# B&R Automation Studio project stopGate_FuB
Automation Studio 4.9

## Logical view

Binary libraries used (declarations not repeated): operator, runtime, astime, AsIecCon, standard

### Package Logical/Libraries - Global libraries

### Library Logical/Libraries/Library (IEC)

#### Library.fun - Exported functions and function blocks
```iecst
{REDUND_ERROR} FUNCTION_BLOCK onOffDebounce (*debounce timer with on delay and off delay capability*) (*$GROUP=User,$CAT=User,$GROUPICON=User.png,$CATICON=User.png*)
	VAR_INPUT
		inputSignal : {REDUND_UNREPLICABLE} BOOL;
		onTimeDelay : {REDUND_UNREPLICABLE} TIME;
		offTimeDelay : {REDUND_UNREPLICABLE} TIME;
	END_VAR
	VAR_OUTPUT
		detected : BOOL;
	END_VAR
	VAR
		onDelayTimer : {REDUND_UNREPLICABLE} TON;
		offDelayTimer : {REDUND_UNREPLICABLE} TOF;
	END_VAR
END_FUNCTION_BLOCK

{REDUND_ERROR} FUNCTION_BLOCK stopGate (*define actuate signal, timeout for gate to open, gate open duration, EMGC input*) (*$GROUP=User,$CAT=User,$GROUPICON=User.png,$CATICON=User.png*)
	VAR_INPUT
		partPresent : {REDUND_UNREPLICABLE} BOOL;
		EMGC : {REDUND_UNREPLICABLE} BOOL;
		gateOpenSensor : {REDUND_UNREPLICABLE} BOOL;
		openTime : {REDUND_UNREPLICABLE} TIME;
		closeTimeout : TIME;
		openTimeout : TIME;
		gateCloseSensor : BOOL;
	END_VAR
	VAR_OUTPUT
		gateOpen : {REDUND_UNREPLICABLE} BOOL;
		sGateOpenFault : {REDUND_UNREPLICABLE} BOOL;
		sGateOpen : {REDUND_UNREPLICABLE} BOOL;
		sGateCloseFault : BOOL;
		gateClose : BOOL;
		sGateClosed : BOOL;
	END_VAR
	VAR
		gateOpenTimeout : {REDUND_UNREPLICABLE} TON;
		state : {REDUND_UNREPLICABLE} INT;
		gateCloseTimeout : TON;
		gateFaultResetTRIG : R_TRIG;
	END_VAR
	VAR_INPUT
		gateFaultReset : BOOL;
		downstreamReady : BOOL;
	END_VAR
	VAR
		partPresentFTRIG : F_TRIG;
		gateOpenTimer : TON;
		gateCloseTimer : TON;
	END_VAR
	VAR_INPUT
		hasOpenSensor : BOOL;
	END_VAR
	VAR
		gateCloseDelay : TON;
		gateCloseDelayTime : TIME;
	END_VAR
END_FUNCTION_BLOCK

{REDUND_ERROR} FUNCTION Timers : BOOL (*Timers used in Automation Line*) (*$GROUP=User,$CAT=User,$GROUPICON=User.png,$CATICON=User.png*)
	VAR_INPUT
		openTimeout : TIME;
		closeTimeout : TIME;
		openTime : TIME;
		closeTime : TIME;
	END_VAR
	VAR
		gateOpenTimeout : TON;
		gateCloseTimeout : TON;
		gateOpenTimer : TON;
		gateCloseTimer : TON;
	END_VAR
	VAR_INPUT
		gateOpen : BOOL;
		gateClose : BOOL;
		gateOpenTimerDone : BOOL;
		gateCloseTImerDone : BOOL;
	END_VAR
END_FUNCTION
```

#### onOffDebounce.st
```iecst
(* debounce timer with on delay and off delay capability *)
FUNCTION_BLOCK onOffDebounce

	onDelayTimer(IN := inputSignal, PT := onTimeDelay);
	detected := onDelayTimer.Q;

	offDelayTimer(IN := detected, PT := offTimeDelay);
	detected := offDelayTimer.Q;

END_FUNCTION_BLOCK
```

#### stopGate.st
```iecst
FUNCTION_BLOCK stopGate

	partPresentFTRIG(CLK := partPresent);  // this indicates that the part has passed by the sensor and the gate is ready to close after
	                                       // a delay timer elapses.

	CASE state OF

		0:  // Starting point of stop gate--everything initialized
			gateOpen := FALSE;
			sGateOpenFault := FALSE;
			sGateCloseFault := FALSE;
			gateOpen := FALSE;
			gateClose := TRUE;
			gateOpenTimeout(IN := FALSE);
			gateCloseTimeout(IN := FALSE);
			gateOpenTimer (IN := FALSE);
			gateCloseTimer (IN := FALSE);
			IF gateCloseSensor THEN
				sGateClosed := TRUE;
				state := 5;
			ELSE
				sGateClosed := FALSE;
				sGateOpen := TRUE ;
				state := 40;
			END_IF

		5:

			// If part arrives at sensor, turn on gateOpen to open gate and move to state 1.  If sensor is used, would
			// need to use de-bounced sensor variable (use onOffDebounce FuB)

			IF partPresent AND downstreamReady AND NOT EMGC THEN  //partPresent would be the .out of onOffDebounce FuB for sensor
				state := 10;
				gateOpen := TRUE;
			END_IF

		10:  // Once gateOpen signal gets triggered, the gate should open within a short time (configurable).  A gate open
			// timeout timer starts at this time.  At this time, if the gate open sensor goes TRUE before the timeout timer
			// matures, then output a signal to signify that the gate is open.  If timer matures and open sensor is still
			// FALSE, then output a gate fault status and move to state 3 where the gate awaits to be fixed, then a "reset"
			// button is pressed to indicate the gate has been fixed.

			gateOpenTimeout(IN := TRUE, PT := openTimeout);
			IF hasOpenSensor THEN

				IF gateOpenSensor THEN
				sGateOpen := TRUE;
				sGateClosed := FALSE;
				state := 20;
				ELSIF gateOpenTimeout.Q THEN
				sGateOpenFault := TRUE;
				sGateOpen := FALSE;
					state := 30;

				END_IF
			ELSE
				state := 20;
			END_IF

		20: // Once in state 20, the gate is known to be opened successfully, and the program waits for the part to
			// pass by the sensor.  Then a closeDelay timer starts.  This timer defines
			// how long the gate should stay open after the falling edge trigger of the sensor
			// goes TRUE (configurable).  When this timer matures, the gateOpen is set TO FALSE which
			// should allow the gate to close, and gateClose is set to TRUE.
			// Once the gateOpen is
			// set to FALSE, a timeout timer similar to state 10 starts timing.  If timer matures and open sensor is still
			// TRUE, then output a gate fault status and move to state 40 where the gate awaits to be fixed, then a "reset"
			// button is pressed to indicate the gate has been fixed.

			// gateOpenTimer (IN := TRUE, PT := openTime);  TODO:  delete if determined not necessary anymore
			gateOpenTimeout (IN := FALSE);

			IF partPresentFTRIG.Q THEN
				gateCloseDelay(IN := TRUE, PT := gateCloseDelayTime);
			END_IF

			IF gateCloseDelay.Q THEN

				gateOpen := FALSE;
				gateClose := TRUE;
				gateCloseTimeout(IN := TRUE, PT := closeTimeout);
				gateCloseDelay(IN := FALSE);
			END_IF

			IF gateCloseSensor THEN
				sGateClosed := TRUE;
				gateCloseTimeout(IN := FALSE);
				state := 0;
				ELSIF gateCloseTimeout.Q THEN
					sGateCloseFault := TRUE;
					sGateClosed := FALSE;
					state := 40;
				END_IF
			END_IF

		30: // Gate Not Open fault reset

			gateFaultResetTRIG(CLK := gateFaultReset);
			gateOpenTimeout (IN := FALSE);

			IF gateFaultResetTRIG.Q THEN
				gateCloseTimeout(IN := FALSE);
				sGateCloseFault := FALSE;
				state := 0;
			END_IF

		40:  // Gate not Closed fault reset

			gateFaultResetTRIG(CLK := gateFaultReset);

			IF gateFaultResetTRIG.Q THEN
				gateCloseTimeout(IN := FALSE);
				sGateCloseFault := FALSE;
				state := 0;
			END_IF

	END_CASE

	IF EMGC THEN
		state := 0;
	END_IF

END_FUNCTION_BLOCK
```

#### Timers.st
```iecst
(* Timers used in Automation Line *)
FUNCTION Timers

END_FUNCTION
```

### Program Logical/ProximityTest (IEC)

#### Variables.var
```iecst
VAR
	inputSignal : BOOL;
	sensor : onOffDebounce;
	onTimeDelay : TIME;
	offTimeDelay : TIME;
	detected : BOOL;
END_VAR
```

#### Cyclic.ld
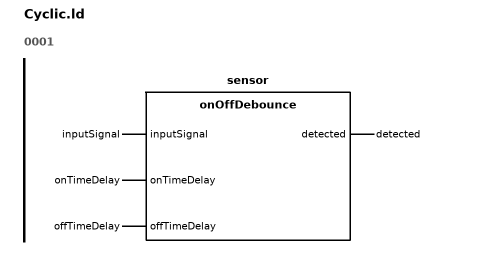
Ladder, written as Structured Text:
```iecst
PROGRAM _CYCLIC
(* Network 1 *)
sensor(inputSignal := inputSignal, onTimeDelay := onTimeDelay, offTimeDelay := offTimeDelay);
detected := sensor.detected;
END_PROGRAM
```

### Program Logical/ProximityTestST (IEC)

#### Variables.var
```iecst
VAR
	sensorST : onOffDebounce;
inputSignal : BOOL;
END_VAR
```

#### Cyclic.st
```iecst
PROGRAM _CYCLIC

	sensorST(inputSignal := inputSignal, onTimeDelay :=T#100ms , offTimeDelay := T#5000ms);

END_PROGRAM
```

### Program Logical/stopGate_TEST (IEC)

#### Variables.var
```iecst
VAR
	partPresent : BOOL;
	gate : stopGate;
	openClose : BOOL;
	EMGC : BOOL;
	gateSensor : BOOL;
	coil : BOOL;
	GATE_FAULT : BOOL;
	GATE_OPEN : BOOL;
	gate1 : stopGate;
	gateOpen : BOOL;
	bladeStopZone0 : ARRAY[0..2] OF stopGate;
	bsZ0partPresent : BOOL;
	gateOpenSensor : BOOL;
	openTime : TIME;
	closeTimeout : TIME;
	openTimeout : TIME;
	hasOpenSensor : BOOL;
	downstreamReady : BOOL;
	gateFaultReset : BOOL;
	gateCloseSensor : BOOL;
	sGateOpenFault : BOOL;
	sGateOpen : BOOL;
	sGateCloseFault : BOOL;
	gateClose : BOOL;
	state : INT;
	sGateClosed : BOOL;
	stopGate_0 : stopGate;
	bladeStopZone1 : stopGate;
END_VAR
```

#### Cyclic.ld
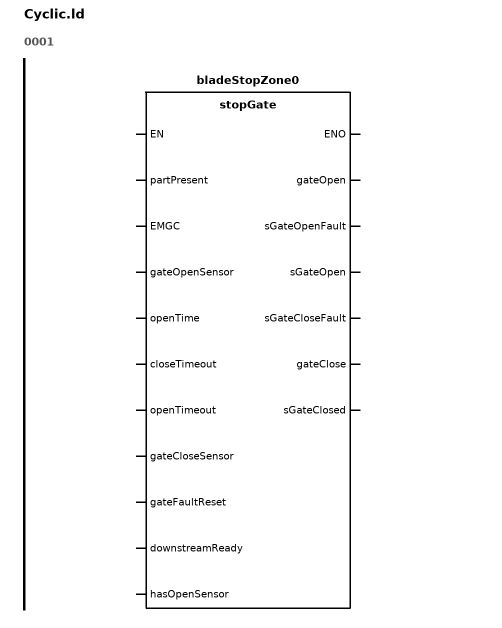
Ladder, written as Structured Text:
```iecst
PROGRAM _CYCLIC
(* Network 1 *)
bladeStopZone0();
END_PROGRAM
```

### Program Logical/FSM/VT_Infeed/VTdispense (IEC)

#### Types.typ
```iecst
TYPE
	vtState :
		(
		New_Member4 := 0,
		New_Member3 := 1,
		New_Member2 := 2,
		New_Member1 := 3,
		New_Member := 4
		);
END_TYPE
```

#### Cyclic.st
```iecst
PROGRAM _CYCLIC

	//**************************************************************************//
	// VT device dispense Control***********************************************//
	// Sept 6, 2024*************************************************************//
	// Jamie Dukelow, Assurant Inc.*********************************************//
	//**************************************************************************//

	//B&R chooses next lane to dispense phone
	// B&R sends signal to VT to dispense phone
	//wait for isDispensing signal
	//once signal is received, increment lane.  if lane not available, increment again
	//if lane still not available, go back to original lane.  if original lane not
	//available, send signal to VT to pause dispensing.  Keep going through this cycle
	//until lane becomes available.  Then resume dispensing.
	//need signal from Transport module as to how many phones are in each lane.

	//Declaring RTrigs

	isDispensingTrig (CLK := isDispensing);
	startTrig(CLK := start);
	errorResetTrig (CLK := errorReset);

	IF laneIdx >=3 THEN  //prevents logic from attempting to dispense into any lane # greater than 2.
		laneIdx := 0;
	END_IF
	// Reset any lane count to zero
	FOR i := 0 TO 2 DO
		resetLaneCountTrig[i] (CLK := resetLaneCount[i]);
		IF resetLaneCountTrig[i].Q THEN
			laneCount[i] := 0;
			resetLaneCount[i] := FALSE;
		END_IF
	END_FOR

	//Resets lane index to 0

	IF startTrig.Q THEN
		laneIdx := 0;
		start := FALSE;
	END_IF

	//doesn't allow dispensing if all lanes are full

	IF (laneCount[0] AND laneCount[1] AND laneCount[2]) >= maxLaneCount THEN
		readyForDispense := FALSE;
	END_IF

	CASE state OF

		0:  //default state

			IF NOT error THEN
				state := 10;
			ELSE
				state := 40;
			END_IF

		10:  //dispense onto lane 0

			IF laneCount[0] < maxLaneCount THEN
				readyForDispense := TRUE;
				laneIdx := 0;
				IF isDispensingTrig.Q THEN
					//laneIdx := laneIdx + 1;
					readyForDispense := FALSE;
					laneCount[0] := laneCount[0] + 1;
					state := 20;
					isDispensing := FALSE;
				END_IF
			ELSE state := 20;
			END_IF

		20: //dispense onto lane 1

			IF laneCount[1] < maxLaneCount THEN
				readyForDispense := TRUE;
				laneIdx := 1;
				IF isDispensingTrig.Q THEN
					readyForDispense := FALSE;
					laneCount[1] := laneCount[1] + 1;
					state := 30;
					isDispensing := FALSE;
				END_IF
			ELSE state := 30;
			END_IF

		30: //dispense onto lane 2

			IF laneCount[2] < maxLaneCount THEN
				readyForDispense := TRUE;
				laneIdx := 2;
				IF isDispensingTrig.Q THEN
					readyForDispense := FALSE;
					laneCount[2] := laneCount[2] + 1;
					state := 10;
					isDispensing := FALSE;
				END_IF
			ELSE state := 0;
			END_IF

		40:  //ERROR state

			IF errorResetTrig.Q THEN
				error := FALSE;
				state := 0;
			ELSE
				state := 40;
			END_IF

	END_CASE

END_PROGRAM

			(*	IF laneIdx = 0 AND NOT downstreamFull AND NOT pauseDispense THEN
					state := 10;
				ELSIF laneIdx = 1 AND NOT downstreamFull AND NOT pauseDispense THEN
					state := 20;
				ELSIF laneIdx = 2 AND NOT downstreamFull AND NOT pauseDispense THEN
					state := 30;
				ELSE state := 0;
				END_IF *)
```

#### Init.st
```iecst
PROGRAM _INIT
	laneIdx := 0;
	readyForDispense := FALSE;
	pauseDispense := FALSE;
	start := FALSE;
	state := 0;
	error := FALSE;

	FOR i := 0 TO 2 DO
		resetLaneCount[i] := FALSE;
		laneCount[i] := 0;
		downstreamFull[i] := FALSE;
	END_FOR

END_PROGRAM
```

### Program Logical/FSM/VT_Infeed/Infeed0 (IEC)

#### Cyclic.st
```iecst
PROGRAM _CYCLIC
	//**************************************************************************//
	// VT--> InfeedZone 0 communications****************************************//
	// Sept 6, 2024*************************************************************//
	// Jamie Dukelow, Assurant Inc.*********************************************//
	//**************************************************************************//

	//Handoff between VT and Infeed Zone 0

	bladeStopZone0();
	partPresent := bladeStopZone0.partPresent;
	gateOpen := bladeStopZone0.gateOpen;
	gateClose := bladeStopZone0.gateClose;
	hasOpenSensor := bladeStopZone0.hasOpenSensor;
	downstreamReady := bladeStopZone0.downstreamReady;
	EMGC := bladeStopZone0.EMGC;

END_PROGRAM
```

### Variables.var
```iecst
VAR
	downstreamFull : ARRAY[0..2] OF BOOL;
	state : INT;
	laneIdx : INT;
	isDispensing : BOOL;
	isDispensingTrig : R_TRIG;
	startTrig : R_TRIG;
	resetLaneCountTrig:  ARRAY[0..2] OF R_TRIG;
	resetLaneCount : ARRAY[0..2] OF BOOL;
	start : BOOL;
	readyForDispense : BOOL;
	error : BOOL;
	errorResetTrig : R_TRIG;
	errorReset : BOOL;
	wrongLane : BOOL; (* if BR requested lane x, and VT dispensed in lane y or z *)
	pauseDispense : BOOL; (* in case all lanes are full *)
	delay : TON;
	laneCount : ARRAY[0..2] OF INT;
	maxLaneCount : INT := 5;
	bladeStopZone0 : stopGate;
	partPresent : BOOL;
	EMGC : BOOL;
	gateOpenSensor : BOOL;
	openTime : TIME;
	closeTimeout : TIME;
	openTimeout : TIME;
	gateCloseSensor : BOOL;
	gateOpen : BOOL;
	sGateOpenFault : BOOL;
	sGateOpen : BOOL;
	sGateCloseFault : BOOL;
	gateClose : BOOL;
	sGateClosed : BOOL;
	gateOpenTimeout : TON;
	gateCloseTimeout : BOOL;
	gateFaultResetTRIG : R_TRIG;
	gateFaultReset : BOOL;
	downstreamReady : BOOL;
	partPresentFTRIG : F_TRIG;
	gateOpenTimer : TON;
	gateCloseTimer : TON;
	hasOpenSensor : BOOL;

	i : INT;

END_VAR

VAR CONSTANT

END_VAR
```

Listed in the project but not available here: Logical/Global.typ, Logical/Global.var, Logical/Libraries/Library/Types.typ, Logical/Libraries/Library/Constants.var, Logical/FSM/VT_Infeed/Types.typ, Logical/FSM/Outfeed, Logical/FSM/Merge, Logical/FSM/Evac
